Staubli VAL3: start.pgx

program start()
  local string l_sVal3
  local string l_sMajor
  local num l_nCtrlPeriod
  local num l_nBoxcarDelay
begin
  logMsg("ros2_server::start : starting application")

  // Get VAL3 version
  l_sVal3=getVersion("System")
  l_sMajor=mid(l_sVal3,1,1)

  // Check boxcar filter configuration
  //$setBoxcarFreq(60.0)
  l_nBoxcarDelay = $getBoxcarDelay()
  logMsg("ros2_server::start : boxcar delay is " + toString("0.1",l_nBoxcarDelay), 1)

  // Speed must be at 100%
  if getMonitorSpeed()<100
    popUpMsg("The monitor speed must be at 100%, waiting...")
    wait(getMonitorSpeed() == 100)
  endIf

  // Reset socket buffers
  clearBuffer(siSocketControl)

  // Setup supervision/diagnostics task
  // TODO

  // Setup control task
  l_nCtrlPeriod = 0.004
  mMdesc.blend = off

  stopMove()
  resetMotion()
  autoConnectMove(true)

  // Start control task
  bIsOverrun = false
  taskCreateSync "controlTask", l_nCtrlPeriod, bIsOverrun, controlTask()
end
